FUNCTION_BLOCK FB_Motor IMPLEMENTS I_Motor
VAR
    bRunning : BOOL := FALSE;
END_VAR

METHOD Start : BOOL
VAR_INPUT
END_VAR
bRunning := TRUE;
Start := bRunning;
END_METHOD

METHOD Stop : BOOL
VAR_INPUT
END_VAR
bRunning := FALSE;
Stop := bRunning;
END_METHOD

END_FUNCTION_BLOCK

(* stored: Version 1.1.0.1, ProductVersion 3.1.4024.16
   POU FB_Motor: Id {87eafeea-6e11-4a4a-b0ac-af4c09b9fc7f}, SpecialFunc None
   Method Start: Id {70aafd24-629a-40d6-af69-fcf362b29eff}
   Method Stop: Id {59c0975e-97ed-4f07-a71b-150155b11fa3} *)
